PROGRAM Zagen
VAR
	MotorUitvoer: BOOL := 0;
	StartZagen: BOOL;
	MotorZagen: BOOL;
	
END_VAR

IF GVL.Power = TRUE THEN 

	
	IF GVL.AanvoerInPositie = TRUE AND StartZagen = TRUE THEN
		MotorZagen :=TRUE;
		GVL.Status:= 'Zaag actief';
		
	END_IF
END_IF

END_PROGRAM

(* stored: Version 1.1.0.1, ProductVersion 3.1.4024.12
   POU Zagen: Id {4c18c0eb-3271-4093-a9fa-bc44a8c4f230}, SpecialFunc None *)
